FUNCTION_BLOCK F_SPLIT_DATE (* split DATE *)
  (* Standard: 61131-3; Classification: standard character and string function; Description: Copyright (c) 2013 TU Wien ACIN and others. This program and the accompanying materials are made available under the terms of the Eclipse Public License 2.0 which is available at https://www.eclipse.org/legal/epl-2.0/ SPDX-License-Identifier: EPL-2.0 Some portions generated by Gemini CLI *)
  (* Version 1.0, 2026-01-31, Franz Höpfinger, HR Agrartechnik GmbH, F_SPLIT_DATE copied from an existing fB and implemented according IEC 61131-3 *)
  PACKAGE iec61131::charString;
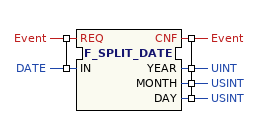
  EVENT_INPUT
    REQ WITH IN; (* Service Request *)
  END_EVENT
  EVENT_OUTPUT
    CNF WITH YEAR, MONTH, DAY; (* Confirmation of Requested Service *)
  END_EVENT
  VAR_INPUT
    IN : DATE; (* Input DATE *)
  END_VAR
  VAR_OUTPUT
    YEAR : UINT; (* Year *)
    MONTH : USINT; (* Month *)
    DAY : USINT; (* Day *)
  END_VAR
  EC_STATES
    REQ : REQ -> CNF;
  END_STATES
  ALGORITHM REQ IN ST:
SPLIT_DATE(IN, YEAR, MONTH, DAY);
  END_ALGORITHM
END_FUNCTION_BLOCK
